Staubli VAL3: readSocket.pgx

program readSocket(num handle_, string& msg_[], bool& result_[])
  local num nChar
  local num nCount
begin
  // read string from socket
  msg_=""
  do
    nCount=sioGet(sSocket[handle_],nChar)
    if (nCount>-1) and (nChar>=32)
      msg_=msg_+chr(nChar)
    endIf
    result_=nCount>-1
    //msg_=sSocket[handle_]
  until (nChar==13) or !result_
  if !result_
    errorCode[handle_]=9
  endIf
  if bDebug
    putln("readStr: "+msg_)
  endIf
end
